TYPE T_PROCESS : DWORD; END_TYPE

(* stored: Version 1.1.0.1
   DUT T_PROCESS: Id {c74bd015-c194-4be6-8b0f-49732c1a216d} *)
